FUNCTION_BLOCK AddRecipeToDatabase
VAR_INPUT
	//BundleData
	//ExtrusionData
	//StrapWrapRecipe
END_VAR
VAR
END_VAR

END_FUNCTION_BLOCK

(* stored: Version 1.1.0.1, ProductVersion 3.1.4024.11
   POU AddRecipeToDatabase: Id {f5939d54-6046-44b2-85b0-95325bce4818}, SpecialFunc None *)
